# EPICS substitutions: rcsRfIoc/rcsRfIocApp/Db/userHost.substitutions
# Example substitutions file

file "db/dbExample1.db" {
    { user = "RCSHost" }
}

file db/dbExample2.db {
    pattern { user, no, scan }
        { "RCSHost", 1, "1 second" }
        { "RCSHost", 2, "2 second" }
        { "RCSHost", 3, "5 second" }
}
